(* This function allows to put ADS strings into the TcUnit ADS message buffer. If Tc2_System.ADSLOGSTR() is used directly,
   the messages can come out of sequence in relation to the message created by TcUnit as TcUnit buffers the messages to
   not overflow the ADS message router. By using this function, the ADS-messages are put in the same buffer as
   TcUnit is using for its output and thus the sequence will be correct *)
FUNCTION TCUNIT_ADSLOGSTR
VAR_INPUT
    msgCtrlMask : DWORD; // Message control mask
    msgFmtStr : Tc2_System.T_MaxString; // Message format string
    strArg : Tc2_System.T_MaxString; // STRING argument
END_VAR

GVL_TcUnit.AdsMessageQueue.WriteLog(MsgCtrlMask := msgCtrlMask,
                                    MsgFmtStr := msgFmtStr,
                                    StrArg := strArg);

END_FUNCTION

(* stored: Version 1.1.0.1, ProductVersion 3.1.4022.18
   POU TCUNIT_ADSLOGSTR: Id {83985386-b582-4673-93b7-d94798f4c9e7}, SpecialFunc None *)
